RoboDK station: Module1-1.rdk

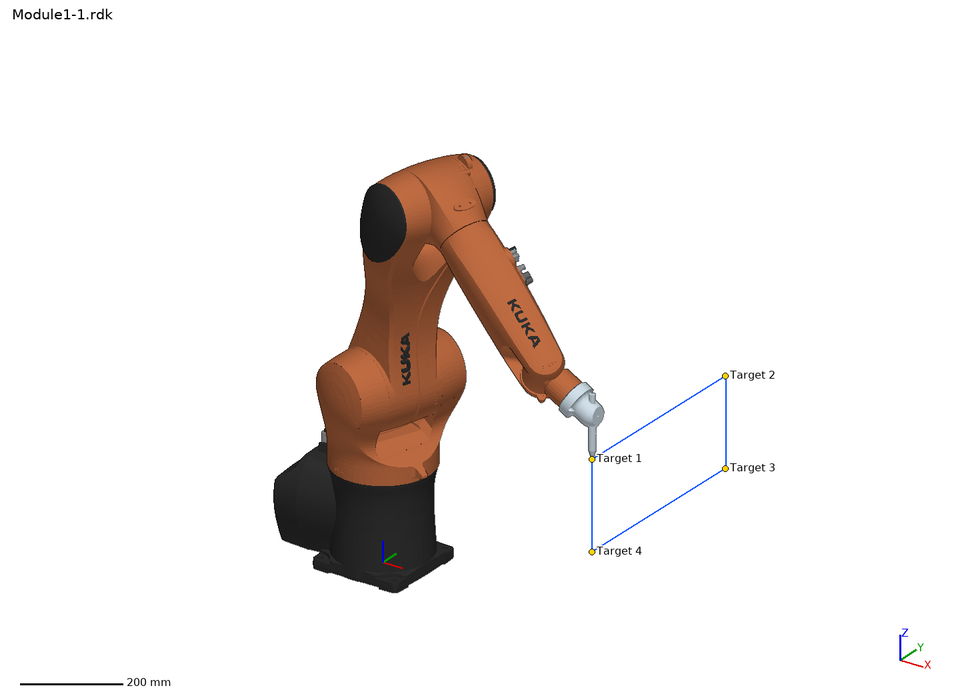
[picture v0: the station drawn from its stored meshes, robots at their saved joint values, targets as dots, program paths as lines]
Station Module1 (saved by RoboDK 5.4.1). Poses are relative to the parent item; angles as X-Y-Z fixed-axis rotations.
Station parameters (name, value as stored): LIN64
  - frame KUKA KR 6 R900 sixx Base at (-207.87, 0, -62.35) mm
    - robot KUKA KR 6 R900 sixx: 6 axes, payload 6 kg, reach 901 mm, repeatability 0.03 mm, weight 52 kg
        modified DH rows (alpha deg, a mm, theta deg, d mm): 0, 0, 0, 400; -90, 25, 0, 0; 0, 455, -90, 0; -90, 35, 0, 420; 90, 0, 0, 0; -90, 0, 180, 80
        joint limits [-170, -190, -120, -185, -120, -350] to [170, 45, 156, 185, 120, 350]; home [0, -90, 90, 0, 0, 0]; saved at [17.23, -74.023, 111.109, 68.718, -15.98, -59.129]
      - tool Pencil, TCP at (82.2, 0, 101.78) mm, rotated rx 0 ry 60 rz 0 deg, size 74.9 x 125 x 107.3 mm
    - target Target 1 (Cartesian target) at (600, -150, 450) mm, rotated rx 180 ry 0 rz -180 deg; joints [17.23, -74.023, 111.109, 68.718, -15.98, -59.129] of KUKA KR 6 R900 sixx
    - target Target 2 (Cartesian target) at (600, 300, 450) mm, rotated rx -180 ry 0 rz 180 deg; joints [-31.81, -67.098, 101.287, -90.006, -27.16, 72.777] of KUKA KR 6 R900 sixx
    - target Target 3 (Cartesian target) at (600, 300, 250) mm, rotated rx -180 ry 0 rz 180 deg; joints [-31.81, -50.164, 108.09, -51.886, -35.464, 28.844] of KUKA KR 6 R900 sixx
    - target Target 4 (Cartesian target) at (600, -150, 250) mm, rotated rx -180 ry 0 rz 180 deg; joints [17.23, -54.835, 118.236, 26.445, -35.172, -13.311] of KUKA KR 6 R900 sixx
  - program Program (7 instructions, listed below)
  - Python program main (listed below)
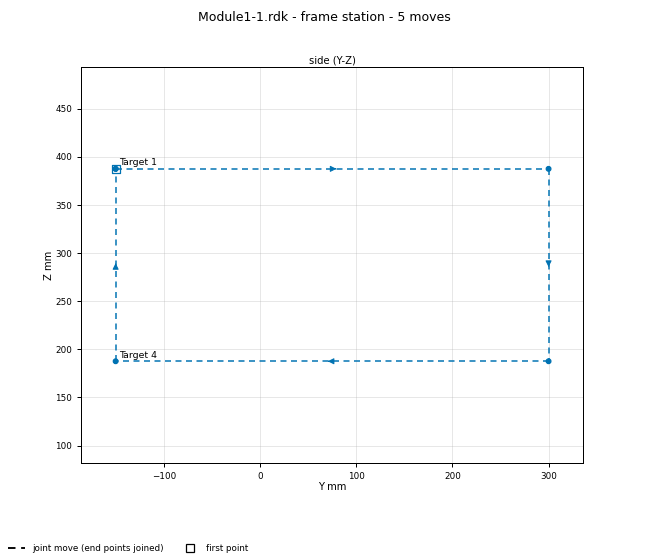
[picture p0: tool path of Module1-1.rdk in frame station, 5 of 5 moves have a stored position in this frame; points joined in program order, loops and branches not executed]

--- program Program (robot KUKA KR 6 R900 sixx) ---
  Set Ref.: KUKA KR 6 R900 sixx Base
  Set Tool: Pencil
  MoveJ (Target 1)
  MoveJ (Target 2)
  MoveJ (Target 3)
  MoveJ (Target 4)
  MoveJ (Target 1)

--- Python program main ---
from robodk.robolink import *      # RoboDK's API
from robodk.robomath import *      # Math toolbox for robots

RL = Robolink()

robot = RL.Item('KUKA KR 6 R900 sixx')

target1 = RL.Item('Target 1')
target2 = RL.Item('Target 2')
target3 = RL.Item('Target 3')
target4 = RL.Item('Target 4')

robot.MoveJ(target1)
robot.MoveJ(target2)
robot.MoveJ(target3)
robot.MoveJ(target4)
robot.MoveJ(target1)
